// TIA Portal V18 export
DATA_BLOCK "Recipe"   // DB76
{ S7_Optimized_Access := 'TRUE' }
VERSION : 0.1
// stored: AutoNumber true, DBAccessibleFromOPCUA true, IsOnlyStoredInLoadMemory false, IsRetainMemResEnabled false, IsWriteProtectedInAS false, MemoryReserve 100
   VAR RETAIN
      RotationStep : Real := 30.0;
   END_VAR
BEGIN
END_DATA_BLOCK
